PROGRAM MAIN
VAR
	cnt : DINT;
END_VAR

cnt := cnt + 1;

END_PROGRAM

(* stored: Version 1.1.0.1, ProductVersion 3.1.4024.12
   POU MAIN: Id {d6de15a2-09c7-4c79-a810-9b276e90cec0}, SpecialFunc None *)
